TYPE (* View rendering style *)
  (* Standard: 61499-1 *)
  (* Version 0.5, 2010-11-01, JHC, Holobloc Inc, Made NONE the initial value. *)
  (* Version 0.4, 2006-04-06, JHC, Holobloc Inc, Added DAMPER. *)
  (* Version 0.3, 2004-09-29, JHC, Rockwell Automation, Added PALLET. *)
  (* Version 0.2, 2002-05-21, JHC, Rockwell Automation, Deleted CLAMP. *)
  (* Version 0.1, 2002-04-25, JHC, Rockwell Automation, Added CLAMP, EMPTY; moved to fb.rt.mva. *)
  (* Version 0.0, 2002-04-01, JHC, Rockwell Automation *)
  (* Compiler header: package fb.rt.dasdA1.A2.Box; *)
  (* Compiler Java Sun JDK 1.4.2 *)
  (* ASN.1 tag PRIVATE 100 *)
  BOXCOLOR : (
    RED,
    YELLOW,
    BLUE
  );
END_TYPE
